// SIMATIC S7-200 project (STEP 7-Micro/WIN), CPU 222 REL 01.22

SYMBOL_TABLE USR1
加泵延时             VW10
减泵延时             VW11
END_SYMBOL_TABLE

ORGANIZATION_BLOCK MAIN:OB1
TITLE=控制工厂车间的水循环冷却系统，为生产设备提供恒压冷却水。系统部署了两台水泵，通过S7-200 PLC控制供水压力保持在设定范围内。涉及的设备包括两台水泵、压力传感器、操作面板按钮和开关，实现较为简单。
// 系统支持两种模式：通过模式选择开关1选择一号泵为主，或通过模式选择开关2选择二号泵为主，以灵活适应不同的运行需求。系统启动时，所有水泵控制信号，包括一号泵变频控制、一号泵工频控制、二号泵变频控制、二号泵工频控制和备用输出，都会被重置，确保进入安全状态。
// 操作员通过模式选择开关决定主泵后，系统优先通过一号泵变频控制或二号泵变频控制让主泵以变频模式运行，实现节能和精确控制。系统会持续监控压力超限传感器。若需要增加供水量，系统通过一号泵工频控制或二号泵工频控制启动辅助泵运行。系统通过模式选择确保一号泵变频控制和二号泵变频控制分时运行，以实现节能控制；系统在状态转移时通过一号泵工频控制或二号泵工频控制单独运行辅助泵，确保供水稳定。
// 若收到加泵信号输入，系统启动加泵延时定时器。延时后，系统进入下一状态以激活辅助泵的工频运行，确保平稳过渡。若压力超限传感器检测到压力过高且一号泵工频控制已置位，系统会通过减泵延时定时器2延时后复位一号泵工频控制，以调整供水量。辅助泵的启动和停止依赖延时定时器，例如工频启动延时定时器1和工频运行延时定时器1，以确保平稳过渡。在压力调节过程中，减泵延时定时器2用于控制辅助泵的停止时机，确保系统平稳运行。
// 系统使用运行状态标志1、运行状态标志2、运行状态标志3和运行状态标志4分步管理运行流程，确保状态有序切换。例如，在一号泵为主模式下，系统从运行状态标志1开始运行一号泵变频控制，根据需求逐步过渡到其他状态，完成循环控制。
BEGIN
Network 1 // 网络标题
// 网络注释
LD     SM0.1
R      Q0.0, 6
R      M0.0, 6
Network 2
// 模式选择：一号泵为主
LD     I0.0
AN     I0.1
CALL   一号泵为主:SBR0
Network 3
// 模式选择：二号泵为主
LD     I0.1
AN     I0.0
CALL   二号泵为主:SBR1
Network 4
// 加、减泵时间赋值
LD     SM0.0
MOVW   +200, 加泵延时:VW10
MOVW   +200, 减泵延时:VW11
Network 5
LD     SM0.0
A      I0.3
AN     T39
TON    T39, 加泵延时:VW10
END_ORGANIZATION_BLOCK

SUBROUTINE_BLOCK 一号泵为主:SBR0
TITLE=子例行程序注释
BEGIN
Network 1 // 网络标题
// 网络注释
LDN    Q0.0
AN     Q0.1
AN     Q0.2
AN     Q0.3
AN     Q0.4
TON    T101, +50
Network 2
LD     T101
EU
S      S0.0, 1
Network 3
LSCR   S0.0
Network 4
// 一号泵变频
LD     SM0.0
LPS
=      Q0.0
A      I0.2
A      Q0.3
A      Q0.0
TON    T40, 减泵延时:VW11
LRD
A      T40
EU
R      Q0.3, 1
LPP
A      T39
AN     Q0.3
EU
SCRT   S0.1
Network 5
SCRE
Network 6
LSCR   S0.1
Network 7
// 一号泵工频
LD     SM0.0
LPS
TON    T41, +5
A      T41
EU
S      Q0.1, 1
LRD
A      Q0.1
TON    T42, +50
LPP
A      T42
EU
SCRT   S0.2
Network 8
SCRE
Network 9
LSCR   S0.2
Network 10
// 2号泵变频
LD     SM0.0
LPS
=      Q0.2
A      I0.2
A      Q0.1
TON    T43, 减泵延时:VW11
LRD
A      T43
EU
R      Q0.1, 1
LPP
A      T39
EU
AN     Q0.1
SCRT   S0.3
Network 11
SCRE
Network 12
LSCR   S0.3
Network 13
// 2号泵工频
LD     SM0.0
LPS
TON    T44, +5
A      T44
EU
S      Q0.3, 1
LRD
A      Q0.3
TON    T45, +50
LPP
A      T45
EU
SCRT   S0.0
Network 14
SCRE
END_SUBROUTINE_BLOCK

SUBROUTINE_BLOCK 二号泵为主:SBR1
TITLE=子例行程序注释
BEGIN
Network 1 // 网络标题
// 网络注释
LDN    Q0.0
AN     Q0.1
AN     Q0.2
AN     Q0.3
AN     Q0.4
TON    T101, +50
Network 2
LD     T101
EU
S      S0.0, 1
Network 3
LSCR   S0.0
Network 4
// 2号泵变频
LD     SM0.0
LPS
=      Q0.2
A      I0.2
A      Q0.1
A      Q0.2
TON    T40, 减泵延时:VW11
LRD
A      T40
EU
R      Q0.1, 1
LPP
A      T39
AN     Q0.1
EU
SCRT   S0.1
Network 5
SCRE
Network 6
LSCR   S0.1
Network 7
// 2号泵工频
LD     SM0.0
LPS
TON    T41, +5
A      T41
EU
S      Q0.3, 1
LRD
A      Q0.3
TON    T42, +50
LPP
A      T42
EU
SCRT   S0.2
Network 8
SCRE
Network 9
LSCR   S0.2
Network 10
// 1号泵变频
LD     SM0.0
LPS
=      Q0.0
A      I0.2
A      Q0.3
TON    T43, 减泵延时:VW11
LRD
A      T43
EU
R      Q0.3, 1
LPP
A      T39
EU
AN     Q0.3
SCRT   S0.3
Network 11
SCRE
Network 12
LSCR   S0.3
Network 13
// 2号泵工频
LD     SM0.0
LPS
TON    T44, +5
A      T44
EU
S      Q0.1, 1
LRD
A      Q0.1
TON    T45, +50
LPP
A      T45
EU
SCRT   S0.0
Network 14
SCRE
Network 20 // 网络标题
// 网络注释
END_SUBROUTINE_BLOCK
